(* IEC 61131-3 sources: CtrlxLadderSkill/tests/features, 7 files *)

(* ---- GVL_IO.st ---- *)
VAR_GLOBAL
    bDI_Start : BOOL;
    bDI_StopOk : BOOL;
    fbGlobalTimer : TON;
END_VAR

(* ---- FB_SimDecl.st ---- *)
// FB_SimDecl: declaration forms the simulator must read. VAR_IN_OUT CONSTANT is a variable
// (no initial values), and based literals (16#...) are constants.
FUNCTION_BLOCK FB_SimDecl
VAR_OUTPUT
    bAbove : BOOL;      // wLevel above LIMIT
END_VAR
VAR_IN_OUT CONSTANT
    wLevel : WORD;      // read-only reference
END_VAR
VAR CONSTANT
    LIMIT : WORD := 16#00FF;
END_VAR

NETWORK Above limit
    [wLevel > LIMIT] -> bAbove
END_FUNCTION_BLOCK

(* ---- FB_SimModels.st ---- *)
// Feature test for ld_sim: struct MOVE copies every member, struct members in compares,
// and an FB box run through a Python model (outputs read back as contacts and via =>).
TYPE ST_Cfg :
STRUCT
    rLimit  : REAL;
    rGain   : REAL;
END_STRUCT
END_TYPE

FUNCTION_BLOCK FB_Child
VAR_INPUT
    bRun    : BOOL;
    rIn     : REAL;
END_VAR
VAR_OUTPUT
    bBusy   : BOOL;
    rOut    : REAL;
END_VAR
bBusy := bRun;
rOut := rIn;
END_FUNCTION_BLOCK

FUNCTION_BLOCK FB_SimModels
VAR_INPUT
    stCfg   : ST_Cfg;
    rValue  : REAL;
    bLatch  : BOOL;
END_VAR
VAR_OUTPUT
    bOver   : BOOL;
    bBusy   : BOOL;
    rChild  : REAL;
END_VAR
VAR
    _stCfg  : ST_Cfg;
    _rScaled : REAL;
    _fbChild : FB_Child;
END_VAR

NETWORK Latch config
    bLatch -> _stCfg := stCfg

NETWORK Scale
    -> _rScaled := MUL(rValue, _stCfg.rGain)

NETWORK Over limit
    [_rScaled > _stCfg.rLimit] -> bOver

NETWORK Child
    -> _fbChild(bRun := bOver, rIn := _rScaled, rOut => rChild)

NETWORK Out bBusy
    _fbChild.bBusy -> bBusy
END_FUNCTION_BLOCK

(* ---- FB_Valve.st ---- *)
FUNCTION_BLOCK FB_Valve
VAR_INPUT
    rSetpoint : REAL;   // setpoint
    bOpen : BOOL;       // command open
END_VAR
VAR_OUTPUT
    eState : INT;       // state
    bOpened : BOOL;     // feedback reached
END_VAR
    eState := 0;
    bOpened := bOpen;
END_FUNCTION_BLOCK

(* ---- ExampleMath.st ---- *)
// Ladder text of references/exports/ctrlx_math_compare.xml (a ctrlX PLC Engineering export).
// tests/run.sh builds it and checks the LD body is element-for-element identical to the export.
PROGRAM ExampleMath
VAR
    in1 : INT;
    in2 : INT;
    out1 : INT;
    out2 : INT;
    out3 : INT;
    out4 : INT;
    equal : BOOL;
    neq : BOOL;
    lessthan : BOOL;
    lessthanorequal : BOOL;
    GreaterThan : BOOL;
    GraterThanOrEqual : BOOL;
END_VAR

NETWORK Addition
    -> out1 := ADD(in1, in2)
NETWORK Subtraction
    -> out2 := SUB(in1, in2)
NETWORK Multiplication
    -> out3 := MUL(in1, in2)
NETWORK Devision
    -> out4 := DIV(in1, in2)
NETWORK Equate
    [out1 = out2] -> equal
NETWORK Not Equal
    [out1 <> out2] -> neq
NETWORK Less Than
    [out1 < out2] -> LessThan
NETWORK Less Than Or Equal TO
    [out1 <= out2] -> LessThanOrEqual
NETWORK Grater Than
    [out1 > out2] -> GreaterThan
NETWORK
    [out1 >= out2] -> GraterThanOrEqual
END_PROGRAM

(* ---- OtherOperators.st ---- *)
// Ladder text of references/exports/ctrlx_other_operators.xml (a ctrlX PLC Engineering export):
// SEL, MUX, LIMIT and a <type>_TO_<type> conversion. tests/run.sh checks the LD body is
// element-for-element identical to the export. (The export mixes In1/in1: CODESYS is case-insensitive.)
PROGRAM OtherOperators
VAR
    bChoice : BOOL;
    In1 : INT;
    In2 : INT;
    out1 : INT;
    iMuxSel : INT;
    in3 : INT;
    in4 : INT;
    in5 : INT;
    out2 : INT;
    minVal : INT;
    maxVal : INT;
    out3 : INT;
    out4 : REAL;
END_VAR

NETWORK Select
    -> out1 := SEL(bChoice, In1, In2)
NETWORK
    -> out2 := MUX(iMuxSel, in1, in2, in3, in4, in5)
NETWORK
    -> out3 := LIMIT(minVal, in3, maxVal)
NETWORK
    -> out4 := INT_TO_REAL(in3)
END_PROGRAM

(* ---- PRG_Conveyor.st ---- *)
// Conveyor written in ladder
PROGRAM PRG_Conveyor
VAR
    bRun : BOOL;              // conveyor running
    bFault : BOOL;
    bReset : BOOL;
    bAuto, bManual, bJog : BOOL;
    fbRunOn : TON;            // run-on timer
    fbCount : CTU;
    afbValve : ARRAY[1..2] OF FB_Valve;
    rTemp : REAL;
    bHot : BOOL;              // decoded compare
    rSp, rOut : REAL;
    iCount : INT;
    tEt : TIME;
END_VAR

NETWORK Start/stop seal-in
// Stop is wired NC, so GVL_IO.bDI_StopOk is TRUE when healthy
    (GVL_IO.bDI_Start | bRun) GVL_IO.bDI_StopOk /bFault -> bRun

NETWORK Run-on delay
    bRun fbRunOn(PT := T#5S, ET => tEt) -> bManual   // trailing comment

NETWORK Count parts
    -> fbCount(CU := bJog, RESET := bReset, PV := 100, Q => bAuto, CV => iCount)

NETWORK
LABEL lblValve
    (bAuto (bJog | /bManual) | bManual N:bJog) -> bJog

NETWORK Hot
// Compares never go in parallel branches: decode first
    [rTemp > 80.0] -> bHot

NETWORK Over-temperature
    (bHot | bFault) /bReset -> S:bFault

NETWORK Setpoint copy
    bAuto -> rOut := rSp, bJog

NETWORK Global timer, unknown-type box
    bRun fbGlobalTimer(PT := T#1S) -> bJog

NETWORK Valve
    -> afbValve[1](rSetpoint := rSp, bOpen := bAuto, eState => iCount, bOpened => bReset)

NETWORK Skip
    bFault -> JMP:lblValve

NETWORK End
    TRUE -> RET
END_PROGRAM
